TYPE Matrix :
STRUCT
	data : ARRAY [0..200,0..200] OF LREAL;
	nRows : INT;
	nCols : INT;
END_STRUCT
END_TYPE

(* stored: Version 1.1.0.1, ProductVersion 3.1.4022.4
   DUT Matrix: Id {ea29ef4f-6b1d-476f-bf4f-2b66d64ab186} *)
